(* IEC 61131-3 sources: CodesysTest/export/Function Blocks/SolenoidValves/FB_DoubleSolenoidClosedCenterActuator.pou/ExtendLPAsserted.prop, 1 file *)

(* ---- Get.pm.st ---- *)
(*#-#-#-#-#-#-#-#-#-#---Declaration---#-#-#-#-#-#-#-#-#-#-#-#-#*)

VAR
END_VAR
(*#-#-#-#-#-#-#-#-#-#---Implementation---#-#-#-#-#-#-#-#-#-#-#-#-#*)

ExtendLPAsserted := solenoid0 AND solenoid1;
